// TIA Portal V20 export
TYPE "typeDataFlinkUsed"
// stored: Access Published, IsFailsafeCompliant true, Namespace Safety
   STRUCT
      CellInterlocks { ExternalWritable := 'False'} : "Safety.s_zc_CellInterlocks";
      NormalInterlocks { ExternalWritable := 'False'} : "Safety.s_zc_NormalInterlocks";
   END_STRUCT;
END_TYPE
